// TIA Portal V18 export
FUNCTION "AHURoomSPActual" : Void   // FC60005, LAD
{ S7_Optimized_Access := 'TRUE' }
VERSION : 0.1
// stored: AutoNumber false, IsIECCheckEnabled false, SetENOAutomatically false, UDAEnableTagReadback false
   VAR_INPUT
      iUnitID : Int;
      rTargetAHUSPTempHeating : Real;
      rTargetAHUSPTempCooling : Real;
      rTargetAHUSPIAQ : Real;
      rTargetAHUSPdP : Real;
   END_VAR
   VAR_OUTPUT
      rActualAHUTempHeatingSP : Real;
      rActualAHUTempCoolingSP : Real;
      rActualAHUIAQSP : Real;
      rActualAHUdPSP : Real;
   END_VAR
   VAR_TEMP
      iTargetUnitMode_old : Int;
      xResetActualOperationMode : Bool;
      iActualUnitMode_old : Int;
      xResetTargetSetpoints : Bool;
   END_VAR
BEGIN

REGION Network 1 (SCL): Smoothing Actual Setpoints
   IF 1 THEN
       #rActualAHUTempHeatingSP := "AHUSetPoints".SetPoints.Room.Target.RATHeating[#iUnitID];
       #rActualAHUTempCoolingSP := "AHUSetPoints".SetPoints.Room.Target.RATCooling[#iUnitID];
       #rActualAHUIAQSP := "AHUSetPoints".SetPoints.Room.Target.IAQ[#iUnitID];
       #rActualAHUdPSP := "AHUSetPoints".SetPoints.Room.Target.BuildingdP[#iUnitID];
   END_IF;
END_REGION
END_FUNCTION
